TYPE uSWversion :
UNION
	a4byte_SWVer 	: 	ARRAY[0..3] OF BYTE;
	UD_SWVer		:	UDINT; 
END_UNION
END_TYPE

(* stored: Version 1.1.0.1, ProductVersion 3.1.4026.18
   DUT uSWversion: Id {d7e2c59d-0566-4f40-ae30-5c4ea1656730} *)
